# EPICS autosave request: iocBoot/ioc13idd_linux/MCB4B_settings.req
# MCB4B motors
file "CARS_motor_settings_sub.req",     P=$(P), M1=m85, M2=m86, M3=m87, M4=m88, M5=m89, M6=m90, M7=m91, M8=m92
